Staubli VAL3: getStandardDeviation.pgx

public program getStandardDeviation(num& x_nInput[], num& x_nStandardDeviation)
  local num l_nVariance
begin

  call getVariance(x_nInput, l_nVariance)

  x_nStandardDeviation = sqrt(l_nVariance)
end
